KUKA KRL program: ho_com_03_ag01_g02.src, ho_com_03_ag01_g02.dat

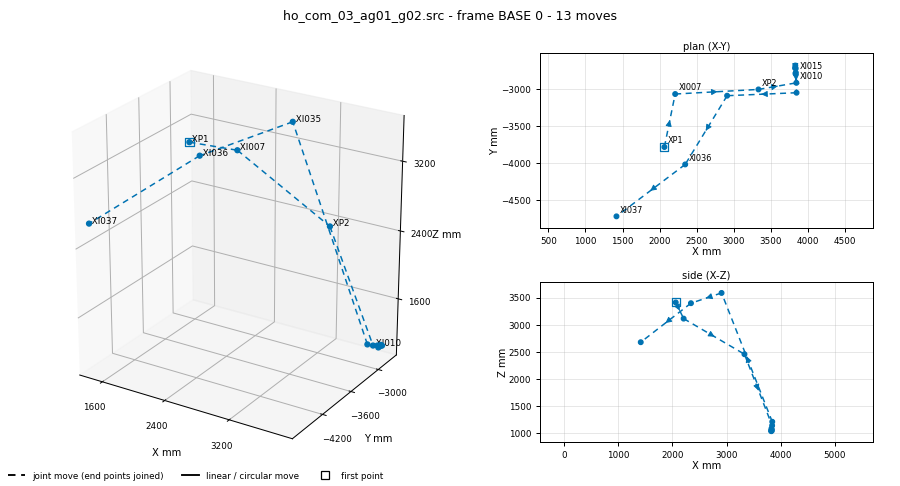
[picture p0: tool path of ho_com_03_ag01_g02.src in frame BASE 0, 13 of 13 moves have a stored position in this frame; points joined in program order, loops and branches not executed]
--- ho_com_03_ag01_g02.src ---
&ACCESS RVO3
&REL 207
&COMMENT Pega Traseira ETB-STB
&PARAM DISKPATH = KRC:\R1\Program\OLP
DEF HO_COM_03_AG01_G02 ( )
;FOLD INI
  ;FOLD BASISTECH INI
    GLOBAL INTERRUPT DECL 3 WHEN $STOPMESS==TRUE DO IR_STOPM ( )
    INTERRUPT ON 3
    BAS (#INITMOV,0)
  ;ENDFOLD (BASISTECH INI)
;FOLD GRIPPERTECH INI
USER_GRP(0,DUMMY,DUMMY,GDEFAULT)
;ENDFOLD (GRIPPERTECH INI)
  ;FOLD USER INI
    ;Make your modifications here

  ;ENDFOLD (USER INI)
;ENDFOLD (INI)

; Caracterizacao dos meios de producao
; Changes: Pega Traseira no AGV
; Modelos: Axor/Atego - ETB/STB
; Versao Atual: 05/01/2016
; Ferramenta: Gripper 913
; Name: P13.050-R1

chk_w11_wechs_ok ( ) ;CHECK GRIPPER 913

;FOLD PTP P1 Vel=100 % PDAT1 Tool[11]:Grp 913 s/ pc Base[0];%{PE}%R 8.2.20,%MKUKATPBASIS,%CMOVE,%VPTP,%P 1:PTP, 2:P1, 3:, 5:100, 7:PDAT1
$BWDSTART=FALSE
PDAT_ACT=PPDAT1
FDAT_ACT=FP1
BAS(#PTP_PARAMS,100)
PTP XP1
;ENDFOLD

;FOLD PULSE 592 'DK 9 GRP Axor 913 Protecao V' State=TRUE CONT Time=1 sec;%{PE}%R 8.2.20,%MKUKATPBASIS,%COUT,%VPULSE,%P 2:592, 3:DK 9 GRP Axor 913 Protecao V, 5:TRUE, 6:CONTINUE, 8:1
CONTINUE
PULSE($OUT[592], TRUE,1)
;ENDFOLD
;FOLD WAIT FOR ( IN 582 'DK 8 GRP Axor 903 Tampa V' AND NOT IN 581 'DK 8 GRP Axor 903 Tampa R' );%{PE}%R 8.2.20,%MKUKATPBASIS,%CEXT_WAIT_FOR,%VEXT_WAIT_FOR,%P 2:, 4:, 5:$IN, 6:582, 7:DK 8 GRP Axor 903 Tampa V, 8:AND, 9:NOT, 10:$IN, 11:581, 12:DK 8 GRP Axor 903 Tampa R, 14:
WAIT FOR  ( $IN[582] AND  NOT $IN[581] )
;ENDFOLD
;FOLD WAIT FOR ( NOT IN 521 'Presença de peça 1 - Axor 913' ) AND ( NOT IN 522 'Presença de peça 2 - Axor 913' );%{PE}%R 8.2.20,%MKUKATPBASIS,%CEXT_WAIT_FOR,%VEXT_WAIT_FOR,%P 2:, 4:NOT, 5:$IN, 6:521, 7:Presença de peça 1 - Axor 913, 9:AND, 10:, 12:NOT, 13:$IN, 14:522, 15:Presença de peça 2 - Axor 913, 17:
WAIT FOR  (  NOT $IN[521] ) AND (  NOT $IN[522] )
;ENDFOLD

;ABRE GRAMPOS
;FOLD SET Z1.1/2 GRP AXOR 913 State=OPN CONT at START Delay=1 ms;%{PE}%R 8.2.1,%MKUKATPGRP,%CGRP,%VGRP,%P 2:10, 4:1, 5:#YES, 6:GDAT10, 8:0, 10:1
TRIGGER WHEN DISTANCE=0 DELAY=1 DO H50(GRP_APO,10,1,GCONT) PRIO=-1
;ENDFOLD
;FOLD SET Z2.1/2 RPS AXOR 913 State=OPN CONT at START Delay=1 ms;%{PE}%R 8.2.1,%MKUKATPGRP,%CGRP,%VGRP,%P 2:11, 4:1, 5:#YES, 6:GDAT11, 8:0, 10:1
TRIGGER WHEN DISTANCE=0 DELAY=1 DO H50(GRP_APO,11,1,GCONT) PRIO=-1
;ENDFOLD
;FOLD SET Z3.1 GRP AXOR 913 State=OPN CONT at START Delay=1 ms;%{PE}%R 8.2.1,%MKUKATPGRP,%CGRP,%VGRP,%P 2:12, 4:1, 5:#YES, 6:GDAT12, 8:0, 10:1
TRIGGER WHEN DISTANCE=0 DELAY=1 DO H50(GRP_APO,12,1,GCONT) PRIO=-1
;ENDFOLD
chk_w11_grp1_opn( )
chk_w11_rps2_opn( )
chk_w11_grp3_opn( )

;FOLD PTP l007 CONT Vel=100 % P_OLP10 Tool[11]:Grp 913 s/ pc Base[0];%{PE}%R 8.2.20,%MKUKATPBASIS,%CMOVE,%VPTP,%P 1:PTP, 2:l007, 3:C_DIS, 5:100, 7:P_OLP10
$BWDSTART=FALSE
PDAT_ACT=PP_OLP10
FDAT_ACT=Fl007
BAS(#PTP_PARAMS,100)
PTP Xl007 C_DIS
;ENDFOLD

;FOLD PTP P2 Vel=100 % PDAT2 Tool[11]:Grp 913 s/ pc Base[0];%{PE}%R 8.2.20,%MKUKATPBASIS,%CMOVE,%VPTP,%P 1:PTP, 2:P2, 3:, 5:100, 7:PDAT2
$BWDSTART=FALSE
PDAT_ACT=PPDAT2
FDAT_ACT=FP2
BAS(#PTP_PARAMS,100)
PTP XP2
;ENDFOLD

; AGUARDA LIBERACAO DE PEGA NO AGV
;FOLD OUT 3370 'Lib. Pegar Painel Traseiro Axor/Atego' State=TRUE ;%{PE}%R 8.2.20,%MKUKATPBASIS,%COUT,%VOUTX,%P 2:3370, 3:Lib. Pegar Painel Traseiro Axor/Atego, 5:TRUE, 6:
$OUT[3370]=TRUE
;ENDFOLD
;FOLD WAIT FOR ( IN 3370 'Lib. p/ Pegar Painel Traseiro Axor/Atego' );%{PE}%R 8.2.20,%MKUKATPBASIS,%CEXT_WAIT_FOR,%VEXT_WAIT_FOR,%P 2:, 4:, 5:$IN, 6:3370, 7:Lib. p/ Pegar Painel Traseiro Axor/Atego, 9:
WAIT FOR  ( $IN[3370] )
;ENDFOLD
;FOLD OUT 3370 'Lib. Pegar Painel Traseiro Axor/Atego' State=FALSE ;%{PE}%R 8.2.20,%MKUKATPBASIS,%COUT,%VOUTX,%P 2:3370, 3:Lib. Pegar Painel Traseiro Axor/Atego, 5:FALSE, 6:
$OUT[3370]=FALSE
;ENDFOLD
;FOLD OUT 3342 'Fora area externa' State=FALSE ;%{PE}%R 8.2.20,%MKUKATPBASIS,%COUT,%VOUTX,%P 2:3342, 3:Fora area externa, 5:FALSE, 6:
$OUT[3342]=FALSE
;ENDFOLD

;FOLD PTP l010 CONT Vel=100 % P_OLP3 Tool[4]:GUN C3 Base[3]:Axor/Atego;%{PE}%R 8.2.20,%MKUKATPBASIS,%CMOVE,%VPTP,%P 1:PTP, 2:l010, 3:C_DIS, 5:100, 7:P_OLP3
$BWDSTART=FALSE
PDAT_ACT=PP_OLP3
FDAT_ACT=Fl010
BAS(#PTP_PARAMS,100)
PTP Xl010 C_DIS
;ENDFOLD
;FOLD LIN l015 CONT Vel=1 m/s CPDAT1 Tool[11]:Grp 913 s/ pc Base[0];%{PE}%R 8.2.20,%MKUKATPBASIS,%CMOVE,%VLIN,%P 1:LIN, 2:l015, 3:C_DIS C_DIS, 5:1, 7:CPDAT1
$BWDSTART=FALSE
LDAT_ACT=LCPDAT1
FDAT_ACT=Fl015
BAS(#CP_PARAMS,1)
LIN Xl015 C_DIS C_DIS
;ENDFOLD
;FOLD LIN l017 CONT Vel=1 m/s CPDAT2 Tool[11]:Grp 913 s/ pc Base[0];%{PE}%R 8.2.20,%MKUKATPBASIS,%CMOVE,%VLIN,%P 1:LIN, 2:l017, 3:C_DIS C_DIS, 5:1, 7:CPDAT2
$BWDSTART=FALSE
LDAT_ACT=LCPDAT2
FDAT_ACT=Fl017
BAS(#CP_PARAMS,1)
LIN Xl017 C_DIS C_DIS
;ENDFOLD

; POSICAO DE PEGA TRASEIRA ETB/STB
;FOLD LIN P_PE06  Vel=0.25 m/s L_OLP1 Tool[11]:Grp 913 s/ pc Base[0];%{PE}%R8.2.19,%MKUKATPBASIS,%CMOVE,%VLIN,%P 1:LIN, 2:P_PE06, 3: , 5:0.25, 7:L_OLP1
$BWDSTART = FALSE
LDAT_ACT= LL_OLP1
FDAT_ACT= FP_PE06
BAS(#CP_PARAMS,0.25)
LIN XP_PE06
;ENDFOLD

IF (NOT(GHOST())) THEN
;FOLD WAIT FOR ( IN 521 'Presença de peça 1 - Axor 913' ) AND ( IN 522 'Presença de peça 2 - Axor 913' );%{PE}%R 8.2.20,%MKUKATPBASIS,%CEXT_WAIT_FOR,%VEXT_WAIT_FOR,%P 2:, 4:, 5:$IN, 6:521, 7:Presença de peça 1 - Axor 913, 9:AND, 10:, 12:, 13:$IN, 14:522, 15:Presença de peça 2 - Axor 913, 17:
WAIT FOR  ( $IN[521] ) AND ( $IN[522] )
;ENDFOLD
ENDIF

; FECHA GRAMPOS
;FOLD SET Z2.1/2 RPS AXOR 913 State=CLO GDAT16;%{PE}%R 8.2.1,%MKUKATPGRP,%CGRP,%VGRP,%P 2:11, 4:2, 5:#NO, 6:GDAT16, 8:0, 10:0
H50(GRP,11,2,GGDAT16)
;ENDFOLD
;FOLD SET Z1.1/2 GRP AXOR 913 State=CLO GDAT4;%{PE}%R 8.2.1,%MKUKATPGRP,%CGRP,%VGRP,%P 2:10, 4:2, 5:#NO, 6:GDAT4, 8:0, 10:0
H50(GRP,10,2,GGDAT4)
;ENDFOLD
;FOLD SET Z3.1 GRP AXOR 913 State=CLO GDAT6;%{PE}%R 8.2.1,%MKUKATPGRP,%CGRP,%VGRP,%P 2:12, 4:2, 5:#NO, 6:GDAT6, 8:0, 10:0
H50(GRP,12,2,GGDAT6)
;ENDFOLD
chk_w11_rps2_clo( )
chk_w11_grp1_clo ( )
chk_w11_grp3_clo ( )

;AGUARDA LIBERACAO SAIR COM PECA
;FOLD OUT 3371 'Lib. p/ sair c/ Traseiro Axor/Atego' State=TRUE ;%{PE}%R 8.2.20,%MKUKATPBASIS,%COUT,%VOUTX,%P 2:3371, 3:Lib. p/ sair c/ Traseiro Axor/Atego, 5:TRUE, 6:
$OUT[3371]=TRUE
;ENDFOLD
;FOLD WAIT FOR ( IN 3371 'Lib. p/ Sair c/ Painel Traseiro Axor/Atego' );%{PE}%R 8.2.20,%MKUKATPBASIS,%CEXT_WAIT_FOR,%VEXT_WAIT_FOR,%P 2:, 4:, 5:$IN, 6:3371, 7:Lib. p/ Sair c/ Painel Traseiro Axor/Atego, 9:
WAIT FOR  ( $IN[3371] )
;ENDFOLD
;FOLD OUT 3371 'Lib. p/ sair c/ Traseiro Axor/Atego' State=FALSE ;%{PE}%R 8.2.20,%MKUKATPBASIS,%COUT,%VOUTX,%P 2:3371, 3:Lib. p/ sair c/ Traseiro Axor/Atego, 5:FALSE, 6:
$OUT[3371]=FALSE
;ENDFOLD

;FOLD LIN l020 Vel=0.25 m/s L_OLP2 Tool[11]:Grp 913 s/ pc Base[0];%{PE}%R 8.2.20,%MKUKATPBASIS,%CMOVE,%VLIN,%P 1:LIN, 2:l020, 3:, 5:0.25, 7:L_OLP2
$BWDSTART=FALSE
LDAT_ACT=LL_OLP2
FDAT_ACT=Fl020
BAS(#CP_PARAMS,0.25)
LIN Xl020
;ENDFOLD

IF (NOT(GHOST())) THEN
;FOLD WAIT FOR ( IN 521 'Presença de peça 1 - Axor 913' ) AND ( IN 522 'Presença de peça 2 - Axor 913' );%{PE}%R 8.2.20,%MKUKATPBASIS,%CEXT_WAIT_FOR,%VEXT_WAIT_FOR,%P 2:, 4:, 5:$IN, 6:521, 7:Presença de peça 1 - Axor 913, 9:AND, 10:, 12:, 13:$IN, 14:522, 15:Presença de peça 2 - Axor 913, 17:
WAIT FOR  ( $IN[521] ) AND ( $IN[522] )
;ENDFOLD
ENDIF

;FOLD PTP l025 CONT Vel=100 % P_OLP5 Tool[12]:Grp 913 c/ pc Base[0];%{PE}%R 8.2.20,%MKUKATPBASIS,%CMOVE,%VPTP,%P 1:PTP, 2:l025, 3:C_DIS, 5:100, 7:P_OLP5
$BWDSTART=FALSE
PDAT_ACT=PP_OLP5
FDAT_ACT=Fl025
BAS(#PTP_PARAMS,100)
PTP Xl025 C_DIS
;ENDFOLD
;FOLD PTP l026 CONT Vel=100 % P_OLP13 Tool[12]:Grp 913 c/ pc Base[0];%{PE}%R 8.2.20,%MKUKATPBASIS,%CMOVE,%VPTP,%P 1:PTP, 2:l026, 3:C_DIS, 5:100, 7:P_OLP13
$BWDSTART=FALSE
PDAT_ACT=PP_OLP13
FDAT_ACT=Fl026
BAS(#PTP_PARAMS,100)
PTP Xl026 C_DIS
;ENDFOLD
;FOLD PTP l035 CONT Vel=100 % P_OLP7 Tool[12]:Grp 913 c/ pc Base[0];%{PE}%R 8.2.20,%MKUKATPBASIS,%CMOVE,%VPTP,%P 1:PTP, 2:l035, 3:C_DIS, 5:100, 7:P_OLP7
$BWDSTART=FALSE
PDAT_ACT=PP_OLP7
FDAT_ACT=Fl035
BAS(#PTP_PARAMS,100)
PTP Xl035 C_DIS
;ENDFOLD
;FOLD PTP l036 CONT Vel=100 % P_OLP11 Tool[12]:Grp 913 c/ pc Base[0];%{PE}%R 8.2.20,%MKUKATPBASIS,%CMOVE,%VPTP,%P 1:PTP, 2:l036, 3:C_DIS, 5:100, 7:P_OLP11
$BWDSTART=FALSE
PDAT_ACT=PP_OLP11
FDAT_ACT=Fl036
BAS(#PTP_PARAMS,100)
PTP Xl036 C_DIS
;ENDFOLD

;LIBERA AREA
;FOLD PULSE 3349 'R1 pegou peça' State=TRUE Time=3 sec;%{PE}%R 8.2.20,%MKUKATPBASIS,%COUT,%VPULSE,%P 2:3349, 3:R1 pegou peça, 5:TRUE, 6:, 8:3
PULSE($OUT[3349], TRUE,3)
;ENDFOLD
;FOLD OUT 3342 'Fora area externa' State=TRUE ;%{PE}%R 8.2.20,%MKUKATPBASIS,%COUT,%VOUTX,%P 2:3342, 3:Fora area externa, 5:TRUE, 6:
$OUT[3342]=TRUE
;ENDFOLD

;FOLD PTP l037 Vel=100 % P_OLP12 Tool[12]:Grp 913 c/ pc Base[0];%{PE}%R 8.2.20,%MKUKATPBASIS,%CMOVE,%VPTP,%P 1:PTP, 2:l037, 3:, 5:100, 7:P_OLP12
$BWDSTART=FALSE
PDAT_ACT=PP_OLP12
FDAT_ACT=Fl037
BAS(#PTP_PARAMS,100)
PTP Xl037
;ENDFOLD

END

--- ho_com_03_ag01_g02.dat ---
&ACCESS RVO3
&REL 207
&COMMENT Pega Traseira ETB-STB
&PARAM DISKPATH = KRC:\R1\Program\OLP
DEFDAT  ho_com_03_ag01_g02
;FOLD EXTERNAL DECLARATIONS;%{PE}%MKUKATPBASIS,%CEXT,%VCOMMON,%P
;FOLD GRIPPERTECH EXT
EXT  H50 (INT  :IN,INT  :IN,INT  :IN,GRP_TYP  :IN )
;ENDFOLD (GRIPPERTECH EXT)
;FOLD SPOTTECH EXT
EXT  USERSPOT (S_COMMAND  :IN,SPOT_TYPE  :IN )
;ENDFOLD (SPOTTECH EXT)
;FOLD BASISTECH EXT;%{PE}%MKUKATPBASIS,%CEXT,%VEXT,%P
EXT  BAS (BAS_COMMAND  :IN,REAL  :IN )
DECL INT SUCCESS
;ENDFOLD (BASISTECH EXT)
;FOLD USER EXT;%{E}%MKUKATPUSER,%CEXT,%VEXT,%P
;Make your modifications here

;ENDFOLD (USER EXT)
;ENDFOLD (EXTERNAL DECLARATIONS)
DECL FDAT Fl010={TOOL_NO 11,BASE_NO 0,IPO_FRAME #BASE,POINT2[] " ",TQ_STATE FALSE}
DECL PDAT PP_OLP3={VEL 100.0,ACC 100.0,APO_DIST 100.0,APO_MODE #CDIS}
DECL E6POS Xl010={X 3841.66699,Y -2916.75488,Z 1144.73401,A -91.1785965,B 65.9535065,C 176.810104,S 2,T 11,E1 -3103.68408,E2 0.0,E3 0.0,E4 0.0,E5 0.0,E6 0.0}
DECL FDAT Fl015={TOOL_NO 11,BASE_NO 0,IPO_FRAME #BASE,POINT2[] " ",TQ_STATE FALSE}
DECL E6POS Xl015={X 3834.60303,Y -2780.03589,Z 1061.80396,A -91.2163391,B 65.3132477,C 176.988297,S 2,T 11,E1 -3103.68604,E2 0.0,E3 0.0,E4 0.0,E5 0.0,E6 0.0}
DECL FDAT FP_PE06={TOOL_NO 11,BASE_NO 0,IPO_FRAME #BASE,POINT2[] " "}
DECL E6POS XP_PE06={X 3827.73291,Y -2683.48096,Z 1041.43799,A -90.5503235,B 66.0767136,C 177.922806,S 2,T 11,E1 -3103.70288,E2 0.0,E3 0.0,E4 0.0,E5 0.0,E6 0.0}
DECL LDAT LL_OLP1={VEL 0.25,ACC 100.0,APO_DIST 0.0,APO_FAC 0.0,ORI_TYP #VAR,CIRC_TYP #BASE,JERK_FAC 50.0}
DECL FDAT Fl020={TOOL_NO 12,BASE_NO 0,IPO_FRAME #BASE,POINT2[] " ",TQ_STATE FALSE}
DECL E6POS Xl020={X 3829.42212,Y -2791.06689,Z 1088.62305,A -91.0449295,B 65.6134186,C 177.290802,S 2,T 11,E1 -3103.68799,E2 0.0,E3 0.0,E4 0.0,E5 0.0,E6 0.0}
DECL LDAT LL_OLP2={VEL 0.25,ACC 100.0,APO_DIST 0.0,APO_FAC 0.0,ORI_TYP #VAR,CIRC_TYP #BASE,JERK_FAC 50.0}
DECL FDAT Fl025={TOOL_NO 12,BASE_NO 0,IPO_FRAME #BASE,POINT2[] " "}
DECL PDAT PP_OLP5={VEL 100.0,ACC 100.0,APO_DIST 10.0,APO_MODE #CDIS}
DECL E6POS Xl025={X 3833.19507,Y -2722.45801,Z 1068.44202,A -91.8144226,B 70.9385529,C 176.583405,S 2,T 11,E1 -3103.68799,E2 0.0,E3 0.0,E4 0.0,E5 0.0,E6 0.0}
DECL FDAT Fl035={TOOL_NO 12,BASE_NO 0,IPO_FRAME #BASE,POINT2[] " "}
DECL PDAT PP_OLP7={VEL 100.0,ACC 100.0,APO_DIST 30.0,APO_MODE #CDIS}
DECL E6POS Xl035={X 2908.521,Y -3090.1499,Z 3592.8269,A -35.5432091,B 49.0769386,C -100.896202,S 2,T 11,E1 -2700.0,E2 0.0,E3 0.0,E4 0.0,E5 0.0,E6 0.0}
DECL BASIS_SUGG_T LAST_BASIS={POINT1[] "P3                      ",POINT2[] "P3                      ",CP_PARAMS[] "CPDAT2                  ",PTP_PARAMS[] "PDAT3                   ",CONT[] "                        ",CP_VEL[] "0.25                    ",PTP_VEL[] "100                     ",SYNC_PARAMS[] "SYNCDAT                 ",SPL_NAME[] "S0                      "}
DECL PDAT PP_OLP10={VEL 100.0,ACC 100.0,APO_DIST 100.0,APO_MODE #CDIS}
DECL E6POS Xl007={X 2208.68311,Y -3067.61304,Z 3118.89307,A -7.49639511,B 64.6939163,C -71.1168518,S 2,T 11,E1 -3169.5791,E2 0.0,E3 0.0,E4 0.0,E5 0.0,E6 0.0}
DECL FDAT Fl007={TOOL_NO 11,BASE_NO 0,IPO_FRAME #BASE,POINT2[] " ",TQ_STATE FALSE}
DECL PDAT PP_OLP11={VEL 100.0,ACC 100.0,APO_DIST 30.0,APO_MODE #CDIS}
DECL E6POS Xl036={X 2343.7229,Y -4016.33789,Z 3403.4729,A -54.7475319,B 53.9433098,C -99.1147385,S 2,T 10,E1 -2700.00098,E2 0.0,E3 0.0,E4 0.0,E5 0.0,E6 0.0}
DECL FDAT Fl036={TOOL_NO 12,BASE_NO 0,IPO_FRAME #BASE,POINT2[] " "}
DECL PDAT PP_OLP12={VEL 100.0,ACC 100.0,APO_DIST 0.0}
DECL E6POS Xl037={X 1417.33105,Y -4716.01904,Z 2683.63989,A -74.2908173,B 82.4296265,C -86.1667709,S 2,T 10,E1 -2912.66699,E2 0.0,E3 0.0,E4 0.0,E5 0.0,E6 0.0}
DECL FDAT Fl037={TOOL_NO 12,BASE_NO 0,IPO_FRAME #BASE,POINT2[] " "}
DECL GRP_SUGG_T LAST_GRP={NUMBER[] "12                      ",STATE[] "2                       ",PARAMS[] "GDAT6                   "}
DECL GRP_TYP GGDAT1={G_APO #NO,GRP_TIME 0.200000003,CTRL #OFF,DLY 0,DST 1}
DECL GRP_TYP GGDAT2={G_APO #NO,GRP_TIME 0.200000003,CTRL #OFF,DLY 0,DST 1}
DECL GRP_TYP GGDAT3={G_APO #NO,GRP_TIME 0.200000003,CTRL #OFF,DLY 0,DST 1}
DECL GRP_TYP GCONT={G_APO #YES,GRP_TIME 0.0,CTRL #OFF,DLY 0,DST 0}
DECL GRP_TYP GGDAT4={G_APO #NO,GRP_TIME 0.200000003,CTRL #OFF,DLY 0,DST 1}
DECL GRP_TYP GGDAT5={G_APO #NO,GRP_TIME 0.200000003,CTRL #OFF,DLY 0,DST 1}
DECL GRP_TYP GGDAT6={G_APO #NO,GRP_TIME 0.200000003,CTRL #OFF,DLY 0,DST 1}
DECL E6POS XP1={X 2063.20703,Y -3781.68994,Z 3417.31299,A -29.1981506,B 53.6340103,C -71.7423782,S 2,T 11,E1 -3170.90308,E2 0.0,E3 0.0,E4 0.0,E5 0.0,E6 0.0}
DECL FDAT FP1={TOOL_NO 11,BASE_NO 0,IPO_FRAME #BASE,POINT2[] " ",TQ_STATE FALSE}
DECL PDAT PPDAT1={VEL 100.0,ACC 80.0,APO_DIST 100.0,APO_MODE #CDIS}
DECL GRP_TYP GGDAT7={G_APO #NO,GRP_TIME 0.200000003,CTRL #OFF,DLY 0,DST 1}
DECL GRP_TYP GGDAT8={G_APO #NO,GRP_TIME 0.200000003,CTRL #OFF,DLY 0,DST 1}
DECL GRP_TYP GGDAT9={G_APO #NO,GRP_TIME 0.200000003,CTRL #OFF,DLY 0,DST 1}
DECL LDAT LCPDAT1={VEL 2.0,ACC 100.0,APO_DIST 10.0,APO_FAC 50.0,AXIS_VEL 100.0,AXIS_ACC 100.0,ORI_TYP #VAR,CIRC_TYP #BASE,JERK_FAC 50.0,GEAR_JERK 50.0,EXAX_IGN 0}
DECL LDAT LCPDAT2={VEL 2.0,ACC 100.0,APO_DIST 10.0,APO_FAC 50.0,AXIS_VEL 100.0,AXIS_ACC 100.0,ORI_TYP #VAR,CIRC_TYP #BASE,JERK_FAC 50.0,GEAR_JERK 50.0,EXAX_IGN 0}
DECL E6POS Xl017={X 3824.16699,Y -2717.20703,Z 1048.51404,A -90.8609314,B 65.8463287,C 177.325195,S 2,T 11,E1 -3103.69507,E2 0.0,E3 0.0,E4 0.0,E5 0.0,E6 0.0}
DECL FDAT Fl017={TOOL_NO 11,BASE_NO 0,IPO_FRAME #BASE,POINT2[] " "}
DECL PDAT PP_OLP13={VEL 100.0,ACC 100.0,APO_DIST 10.0,APO_MODE #CDIS}
DECL E6POS Xl026={X 3844.15308,Y -3050.0769,Z 1215.58398,A -91.8146591,B 70.9384689,C 176.582993,S 2,T 11,E1 -3103.68896,E2 0.0,E3 0.0,E4 0.0,E5 0.0,E6 0.0}
DECL FDAT Fl026={TOOL_NO 12,BASE_NO 0,IPO_FRAME #BASE,POINT2[] " "}
DECL GRP_TYP GGDAT10={G_APO #NO,GRP_TIME 0.200000003,CTRL #OFF,DLY 0,DST 1}
DECL GRP_TYP GGDAT11={G_APO #NO,GRP_TIME 0.200000003,CTRL #OFF,DLY 0,DST 1}
DECL GRP_TYP GGDAT12={G_APO #NO,GRP_TIME 0.200000003,CTRL #OFF,DLY 0,DST 1}
DECL GRP_TYP GGDAT13={G_APO #NO,GRP_TIME 0.200000003,CTRL #OFF,DLY 0,DST 1}
DECL GRP_TYP GGDAT14={G_APO #NO,GRP_TIME 0.200000003,CTRL #OFF,DLY 0,DST 1}
DECL GRP_TYP GGDAT15={G_APO #NO,GRP_TIME 0.200000003,CTRL #OFF,DLY 0,DST 1}
DECL GRP_TYP GGDAT16={G_APO #NO,GRP_TIME 0.200000003,CTRL #OFF,DLY 0,DST 1}
DECL E6POS XP2={X 3331.12109,Y -3005.60498,Z 2462.18896,A -59.7037086,B 70.3952103,C -135.742203,S 2,T 11,E1 -3134.22192,E2 0.0,E3 0.0,E4 0.0,E5 0.0,E6 0.0}
DECL FDAT FP2={TOOL_NO 11,BASE_NO 0,IPO_FRAME #BASE,POINT2[] " ",TQ_STATE FALSE}
DECL PDAT PPDAT2={VEL 100.0,ACC 100.0,APO_DIST 100.0,APO_MODE #CDIS}
DECL E6POS XP3={X 6395.78516,Y -5593.32324,Z -181.380096,A -0.626903117,B -65.7444611,C -10.01227,S 2,T 11,E1 -3104.37891,E2 0.0,E3 0.0,E4 0.0,E5 0.0,E6 0.0}
DECL FDAT FP3={TOOL_NO 4,BASE_NO 3,IPO_FRAME #BASE,POINT2[] " ",TQ_STATE FALSE}
DECL PDAT PPDAT3={VEL 100.0,ACC 100.0,APO_DIST 100.0,APO_MODE #CDIS}
ENDDAT
